FUNCTION_BLOCK FB_Motion
VAR_IN_OUT

/// axis reference data structure 
	Master: AXIS_REF;
	/// axis reference data structure 
	Slave: AXIS_REF;
	PowerMaster: MC_Power;
	PowerSlave: MC_Power;
	GO : BOOL;// := FALSE;
END_VAR
VAR_OUTPUT
END_VAR
VAR

	/// state machine state 
	state: MoveState_t;
	
	/// debug function block output data 
	PowerMasterOut: ST_McOutputs;
	
	/// debug function block output data 
	PowerSlaveOut: ST_McOutputs;
	//MoveMaster: MC_MoveAbsolute;
	/// debug function block output data 
	MoveMasterOut: ST_McOutputs;
	//MoveSlave: MC_MoveAbsolute;
	/// debug function block output data 
	MoveSlaveOut: ST_McOutputs;
	ResetMaster: MC_Reset;
	/// debug function block output data 
	ResetMasterOut: ST_McOutputs;
	ResetSlave: MC_Reset;
	/// debug function block output data 
	ResetSlaveOut: ST_McOutputs;
	GearIn: MC_GearIn;
	GearInOut: ST_McOutputs;
	GearOut: MC_GearOut;
	GearOutOut: ST_McOutputs;
	HaltSlave: MC_Halt;
	HaltSlaveOut: ST_McOutputs;
	
	MoveMaster: MC_MoveRelative;
	MoveSlave: MC_MoveRelative;
END_VAR

	(* update the axis status at the beginning of each cycle *)
	//Master();
	//Slave();
if  NOT (GO) then
	state := MOVESTATE_INIT;	
END_IF
	(* move axis using a state machine *)
	CASE state OF

		MOVESTATE_INIT :	(* initialisation *)
			(* initialize all function blocks *)
			MoveMaster.Execute := FALSE;
			MoveSlave.Execute := FALSE;
			HaltSlave.Execute := FALSE;
			ResetMaster.Execute := FALSE;
			ResetSlave.Execute := FALSE;
			GearIn.Execute := FALSE;
			GearOut.Execute := FALSE;
			if (GO) then
				state := MOVESTATE_ENABLE;	
			END_IF
			

		MOVESTATE_ENABLE :
		//	PowerMaster.Enable := TRUE;
		//	PowerMaster.Enable_Positive := TRUE;
		//	PowerMaster.Enable_Negative := TRUE;
		//	PowerSlave.Enable := TRUE;
		//	PowerSlave.Enable_Positive := TRUE;
		//	PowerSlave.Enable_Negative := TRUE;
			IF PowerMaster.Status AND PowerSlave.Status THEN
				state := MOVESTATE_COUPLE;
			ELSIF PowerMaster.Error OR PowerSlave.Error THEN
				state := MOVESTATE_ERROR;
			END_IF

		MOVESTATE_COUPLE :
			GearIn.Execute := TRUE;
			IF GearIn.InGear THEN
				GearIn.Execute := FALSE;
				state := MOVESTATE_FORWARD1;
			ELSIF GearIn.Error THEN
				state := MOVESTATE_ERROR;
			END_IF

		MOVESTATE_FORWARD1:		(* start to first position *)
			MoveMaster.Distance := 7;		(* start to intermediate target position *)
			MoveMaster.Velocity := 0.3;		(* medium velocity level *)
			MoveMaster.BufferMode := MC_Buffered;
			MoveMaster.Execute := TRUE;
			IF Master.NcToPlc.SetPos > 20 THEN
				state := MOVESTATE_HALTSLAVE;
			ELSIF MoveMaster.Done  THEN
				(* axis is executing job but is not yet finished *)
				MoveMaster.Execute := FALSE;
				state := MOVESTATE_BACKWARDS;
			ELSIF MoveMaster.CommandAborted OR MoveMaster.Error THEN
				state := MOVESTATE_ERROR;
			END_IF

		MOVESTATE_HALTSLAVE :
			(* stopping a slave in motion is possible from TwinCAT 2.11if
			    the parameter "allow motion commands to slaves" is enabled.
			    The slave will automatically be decoupled and stoped.
			*)
			HaltSlave.Execute := TRUE;
			IF HaltSlave.Done AND MoveMaster.Done THEN (* wait for master and slave finished *)
				MoveMaster.Execute := FALSE;
				HaltSlave.Execute := FALSE;
				state := MOVESTATE_COUPLE2;
			ELSIF HaltSlave.Error OR HaltSlave.CommandAborted THEN
				state := MOVESTATE_ERROR;
			ELSIF MoveMaster.CommandAborted OR MoveMaster.Error THEN
				state := MOVESTATE_ERROR;
			END_IF

		MOVESTATE_COUPLE2 :
			GearIn.Execute := TRUE;
			IF GearIn.InGear THEN
				GearIn.Execute := FALSE;
				state := MOVESTATE_FORWARD2;
			ELSIF GearIn.Error THEN
				state := MOVESTATE_ERROR;
			END_IF

		MOVESTATE_FORWARD2 :			(* move to next position *)
			MoveMaster.Distance := 5;		(* start to target position *)
			MoveMaster.Velocity := 0.2;		(* medium velocity level *)
			MoveMaster.BufferMode := MC_Buffered;
			MoveMaster.Execute := TRUE;
			IF Master.NcToPlc.SetPos > 25 THEN
				state := MOVESTATE_DECOUPLE;
			ELSIF MoveMaster.Done  THEN
				(* axis is executing job but is not yet finished *)
				MoveMaster.Execute := FALSE;
				state := MOVESTATE_BACKWARDS;
			ELSIF MoveMaster.CommandAborted OR MoveMaster.Error THEN
				state := MOVESTATE_ERROR;
			END_IF

		MOVESTATE_DECOUPLE :
			(* if a slave is decoupled in motion the axis will continue moving at constant velocity *)
			GearOut.Execute := TRUE;
			IF GearOut.Done AND MoveMaster.Done THEN (* wait for master motion finished *)
				GearOut.Execute := FALSE;
				MoveMaster.Execute := FALSE;
				state := MOVESTATE_BACKWARDS;
			ELSIF GearOut.Error THEN
				state := MOVESTATE_ERROR;
			ELSIF MoveMaster.CommandAborted OR MoveMaster.Error THEN
				state := MOVESTATE_ERROR;
			END_IF

		MOVESTATE_BACKWARDS :	(* move back to initial position *)
			MoveMaster.Distance := -12;		(* position close to initial position *)
			MoveMaster.Velocity := 0.3;		(* high velocity *)
			MoveMaster.Execute := TRUE;
			MoveSlave.Distance := -10;		(* position close to initial position *)
			MoveSlave.Velocity := 0.3;		(* high velocity *)
			MoveSlave.Execute := TRUE;
			IF MoveMaster.Done AND MoveSlave.Done THEN
				(* axis is executing job but is not yet finished *)
				MoveMaster.Execute := FALSE;
				(* leave this state and buffer a second command *)
				state := MOVESTATE_INIT;
			ELSIF MoveMaster.CommandAborted OR MoveMaster.Error
				OR  MoveSlave.CommandAborted OR MoveSlave.Error
				THEN
				state := MOVESTATE_ERROR;
			END_IF

		MOVESTATE_ERROR :
			IF Master.Status.Error OR Slave.Status.Error THEN
				state := MOVESTATE_RESET;	(* axis error requires reset *)
			ELSE
				state := MOVESTATE_INIT;		(* function block errors don't need a reset *)
			END_IF

		MOVESTATE_RESET :
			ResetMaster.Execute := TRUE;
			ResetSlave.Execute := TRUE;
			IF ResetMaster.Done AND ResetSlave.Done THEN
				state := MOVESTATE_INIT;
			ELSIF ResetMaster.Error OR ResetSlave.Error THEN
				state := MOVESTATE_INIT; (* can't do anything here *)
			END_IF

	END_CASE

	//ActPower();		(* call the power function block *)
	ActMoveRel();		(* call the move function block *)
	ActReset();		(* call the reset function block *)
	ActCouple();		(* call the master slave coupling function block *)

ACTION ActCouple:
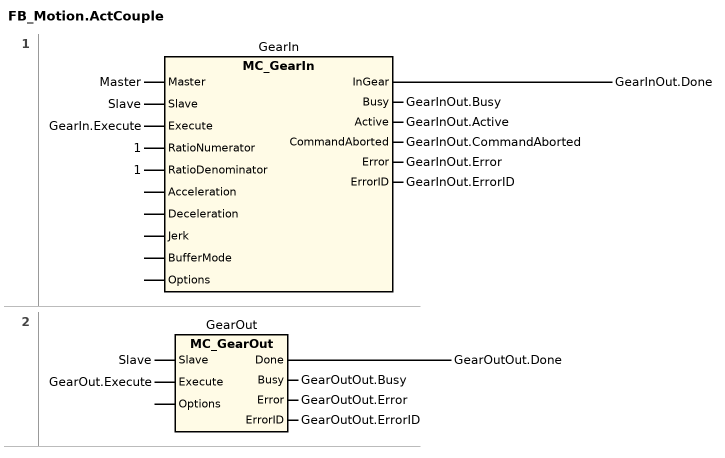
// NETWORK 1
GearIn(
    Master := Master,
    Slave := Slave,
    Execute := GearIn.Execute,
    RatioNumerator := 1,
    RatioDenominator := 1,
    Busy => GearInOut.Busy,
    Active => GearInOut.Active,
    CommandAborted => GearInOut.CommandAborted,
    Error => GearInOut.Error,
    ErrorID => GearInOut.ErrorID); // MC_GearIn
GearInOut.Done := GearIn.InGear;

// NETWORK 2
GearOut(
    Slave := Slave,
    Execute := GearOut.Execute,
    Busy => GearOutOut.Busy,
    Error => GearOutOut.Error,
    ErrorID => GearOutOut.ErrorID); // MC_GearOut
GearOutOut.Done := GearOut.Done;
END_ACTION

ACTION ActMove:
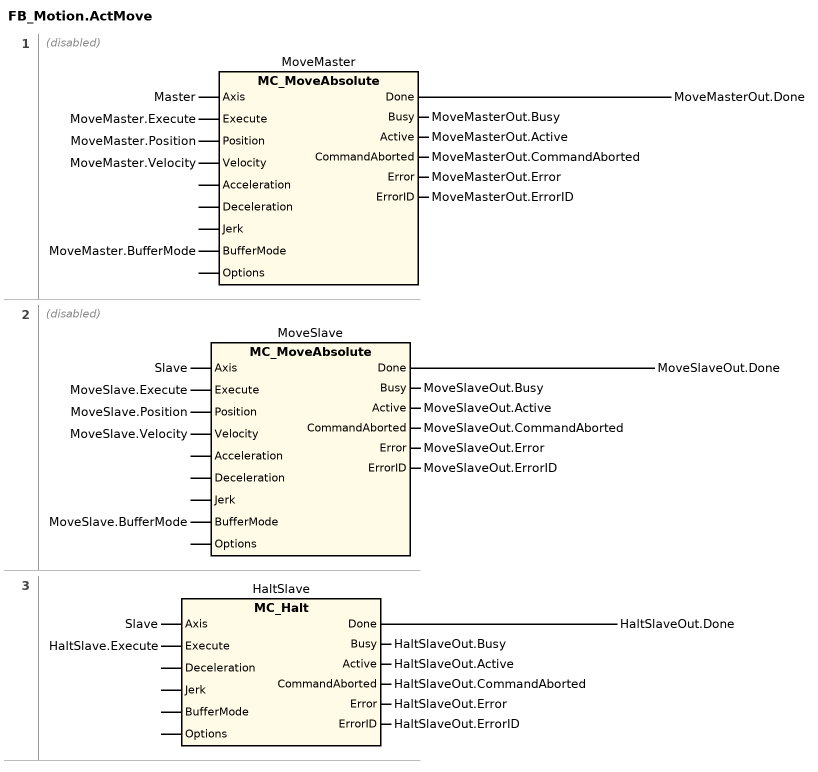
// NETWORK 1 (disabled)
// MoveMaster(
//     Axis := Master,
//     Execute := MoveMaster.Execute,
//     Position := MoveMaster.Position,
//     Velocity := MoveMaster.Velocity,
//     BufferMode := MoveMaster.BufferMode,
//     Busy => MoveMasterOut.Busy,
//     Active => MoveMasterOut.Active,
//     CommandAborted => MoveMasterOut.CommandAborted,
//     Error => MoveMasterOut.Error,
//     ErrorID => MoveMasterOut.ErrorID); // MC_MoveAbsolute
// MoveMasterOut.Done := MoveMaster.Done;

// NETWORK 2 (disabled)
// MoveSlave(
//     Axis := Slave,
//     Execute := MoveSlave.Execute,
//     Position := MoveSlave.Position,
//     Velocity := MoveSlave.Velocity,
//     BufferMode := MoveSlave.BufferMode,
//     Busy => MoveSlaveOut.Busy,
//     Active => MoveSlaveOut.Active,
//     CommandAborted => MoveSlaveOut.CommandAborted,
//     Error => MoveSlaveOut.Error,
//     ErrorID => MoveSlaveOut.ErrorID); // MC_MoveAbsolute
// MoveSlaveOut.Done := MoveSlave.Done;

// NETWORK 3
HaltSlave(
    Axis := Slave,
    Execute := HaltSlave.Execute,
    Busy => HaltSlaveOut.Busy,
    Active => HaltSlaveOut.Active,
    CommandAborted => HaltSlaveOut.CommandAborted,
    Error => HaltSlaveOut.Error,
    ErrorID => HaltSlaveOut.ErrorID); // MC_Halt
HaltSlaveOut.Done := HaltSlave.Done;
END_ACTION

ACTION ActMoveRel:
MoveMaster(
	Axis:= Master , 
	Execute:= , 
	Distance:= , 
	Velocity:= , 
	Acceleration:= , 
	Deceleration:= , 
	Jerk:= , 
	BufferMode:= , 
	Options:= , 
	Done=> MoveMasterOut.Done, 
	Busy=> MoveMasterOut.Busy, 
	Active=> MoveMasterOut.Active , 
	CommandAborted=> MoveMasterOut.CommandAborted , 
	Error=> MoveMasterOut.Error, 
	ErrorID=> MoveMasterOut.ErrorID );
	
MoveSlave(
	Axis:= Slave, 
	Execute:= , 
	Distance:= , 
	Velocity:= , 
	Acceleration:= , 
	Deceleration:= , 
	Jerk:= , 
	BufferMode:= , 
	Options:= , 
	Done=> MoveSlaveOut.Done, 
	Busy=> MoveSlaveOut.Busy, 
	Active=> MoveSlaveOut.Active , 
	CommandAborted=> MoveSlaveOut.CommandAborted , 
	Error=> MoveSlaveOut.Error, 
	ErrorID=> MoveSlaveOut.ErrorID );
END_ACTION

ACTION ActPower:
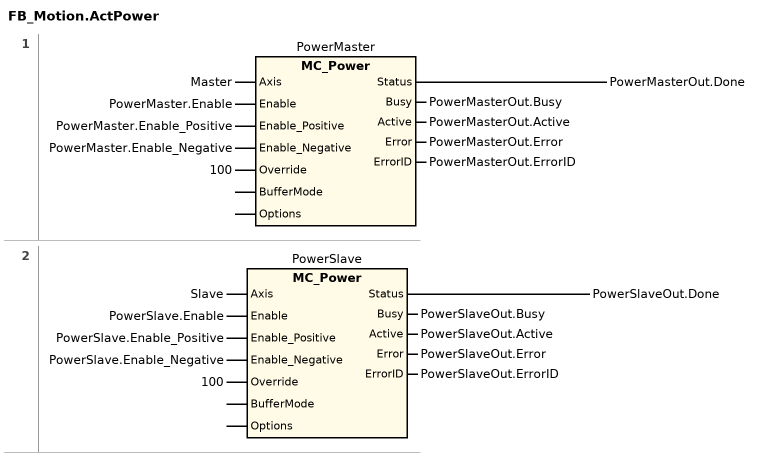
// NETWORK 1
PowerMaster(
    Axis := Master,
    Enable := PowerMaster.Enable,
    Enable_Positive := PowerMaster.Enable_Positive,
    Enable_Negative := PowerMaster.Enable_Negative,
    Override := 100,
    Busy => PowerMasterOut.Busy,
    Active => PowerMasterOut.Active,
    Error => PowerMasterOut.Error,
    ErrorID => PowerMasterOut.ErrorID); // MC_Power
PowerMasterOut.Done := PowerMaster.Status;

// NETWORK 2
PowerSlave(
    Axis := Slave,
    Enable := PowerSlave.Enable,
    Enable_Positive := PowerSlave.Enable_Positive,
    Enable_Negative := PowerSlave.Enable_Negative,
    Override := 100,
    Busy => PowerSlaveOut.Busy,
    Active => PowerSlaveOut.Active,
    Error => PowerSlaveOut.Error,
    ErrorID => PowerSlaveOut.ErrorID); // MC_Power
PowerSlaveOut.Done := PowerSlave.Status;
END_ACTION

ACTION ActReset:
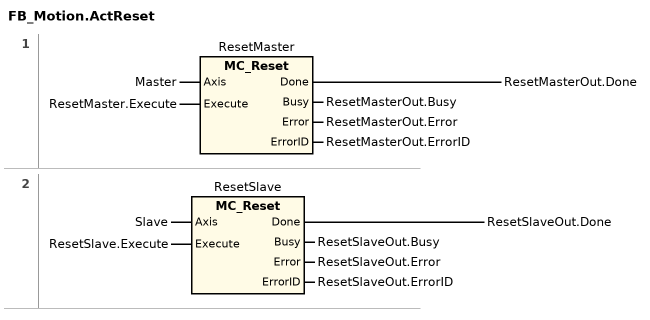
// NETWORK 1
ResetMaster(
    Axis := Master,
    Execute := ResetMaster.Execute,
    Busy => ResetMasterOut.Busy,
    Error => ResetMasterOut.Error,
    ErrorID => ResetMasterOut.ErrorID); // MC_Reset
ResetMasterOut.Done := ResetMaster.Done;

// NETWORK 2
ResetSlave(
    Axis := Slave,
    Execute := ResetSlave.Execute,
    Busy => ResetSlaveOut.Busy,
    Error => ResetSlaveOut.Error,
    ErrorID => ResetSlaveOut.ErrorID); // MC_Reset
ResetSlaveOut.Done := ResetSlave.Done;
END_ACTION

END_FUNCTION_BLOCK

(* stored: Version 1.1.0.1, ProductVersion 3.1.4022.12
   POU FB_Motion: Id {3d36cdba-609d-4c8d-b14f-82d0e9d5ddc5}, SpecialFunc None
   Action ActCouple: Id {1ea7a302-82ed-4cb8-ab5b-5068e50825ec}
   Action ActMove: Id {24910667-1ea8-43aa-bc38-0ac08d39f462}
   Action ActMoveRel: Id {77d7c459-bca9-4368-98fe-8b84702ad28b}
   Action ActPower: Id {cd1a3896-ea57-4bf3-9744-5a49b63cbbda}
   Action ActReset: Id {2bce11ae-74a8-4b01-b730-0d6603b9dc9e} *)
